// TwinCAT 3 PLC project RTNNI
// Title: Real-Time Neural Network generator
// Company: ISW
// Author: Zexu Zhou, Christoph Hinze
// ProjectVersion: 0.1
// ProgramVersion: 3.1.4024.0
// libraries:
//   Tc2_Standard, * (Beckhoff Automation GmbH)
//   Tc2_System, * (Beckhoff Automation GmbH)
//   Tc2_Utilities, * (Beckhoff Automation GmbH)
//   Tc3_Module, * (Beckhoff Automation GmbH)
// project tree:
//   DUTs/ act_type.TcDUT (not stored), Dense_v1_Layers.TcDUT, Dense_v1_LayerWeights.TcDUT, Layer.TcDUT (not stored), norm_type.TcDUT
//   / PlcTask.TcTTO
//   POUs/activation function/ F_exponential.TcPOU (not stored), F_relu.TcPOU (not stored), F_selu.TcPOU, F_sigmoid.TcPOU (not stored), F_silu.TcPOU (not stored), F_softplus.TcPOU, F_softsign.TcPOU (not stored), F_tanh.TcPOU
//   POUs/ FB_Dense_v1.TcPOU, FB_LoadWeights.TcPOU, F_ForwardPropagation.TcPOU (not stored), MAIN.TcPOU
//   POUs/math/ F_Dot.TcPOU (not stored)
//   POUs/normalization/ F_denormalization.TcPOU (not stored), F_normalization.TcPOU (not stored), F_NormalizationLayer.TcPOU

CONFIGURATION RTNNI
    RESOURCE PLC ON TwinCAT3
        TASK PlcTask(INTERVAL := T#10ms, PRIORITY := 21);
        PROGRAM MAIN WITH PlcTask : MAIN;
    END_RESOURCE
END_CONFIGURATION

// ---- DUTs/Dense_v1_Layers.TcDUT
TYPE Dense_v1_Layers:
STRUCT
    num_layers : UINT := 5;
    weights : Dense_v1_LayerWeights;
    layers : ARRAY[0..4] OF Layer :=[
    (num_neurons := 5),
    (num_neurons := 100, activation := act_type.relu, pointer_weight:= ADR(weights.HiddenLayers1_weight),pointer_bias:= ADR(weights.HiddenLayers1_bias)),
    (num_neurons := 100, activation := act_type.relu, pointer_weight:= ADR(weights.HiddenLayers2_weight),pointer_bias:= ADR(weights.HiddenLayers2_bias)),
    (num_neurons := 100, activation := act_type.relu, pointer_weight:= ADR(weights.HiddenLayers3_weight),pointer_bias:= ADR(weights.HiddenLayers3_bias)),
    (num_neurons := 1,activation := act_type.linear, normalization := norm_type.denormalization, pointer_weight:= ADR(weights.OutputLayer_weight),pointer_bias:= ADR(weights.OutputLayer_bias))];
    layer_output : ARRAY[0..99] OF LREAL;
    layer_input : ARRAY[0..99] OF LREAL;
    
END_STRUCT
END_TYPE

// ---- DUTs/Dense_v1_LayerWeights.TcDUT
TYPE Dense_v1_LayerWeights:
STRUCT
    normalization_mean : ARRAY[0..0] OF LREAL;
    normalization_std : ARRAY[0..0] OF LREAL;
    HiddenLayers1_weight : ARRAY[0..99,0..4] OF LREAL;
    HiddenLayers1_bias : ARRAY[0..99] OF LREAL;
    HiddenLayers2_weight : ARRAY[0..99,0..99] OF LREAL;
    HiddenLayers2_bias : ARRAY[0..99] OF LREAL;
    HiddenLayers3_weight : ARRAY[0..99,0..99] OF LREAL;
    HiddenLayers3_bias : ARRAY[0..99] OF LREAL;
    OutputLayer_weight : ARRAY[0..0,0..99] OF LREAL;
    OutputLayer_bias : ARRAY[0..0] OF LREAL;
    denormalization_mean : ARRAY[0..0] OF LREAL;
    denormalization_std : ARRAY[0..0] OF LREAL;
    hash_sha_256 : ARRAY[0..3] OF LREAL;
END_STRUCT
END_TYPE

// ---- DUTs/norm_type.TcDUT
{attribute 'qualified_only'}
{attribute 'strict'}
TYPE norm_type :
(	
	none := 0,	
	normalization := 1,
	denormalization :=2
);
END_TYPE

// ---- POUs/MAIN.TcPOU
PROGRAM MAIN
VAR
	input : ARRAY[0..4] OF LREAL := [1,1,1,1,1];	
	out : ARRAY[0..0] OF LREAL;
	FB_NN : FB_Dense_v1;
	
	test_in : LREAL := 50;
	test_flg : BOOL := FALSE;
END_VAR

FB_NN(pointer_input := ADR(input),pointer_output:= ADR(out));
IF NOT test_flg THEN
	F_NormalizationLayer(pointer_input := ADR(test_in),pointer_mean := ADR(FB_NN.nn.weights.denormalization_mean),
	pointer_std := ADR(FB_NN.nn.weights.denormalization_std),invert := TRUE, num_neurons := FB_NN.nn.layers[SIZEOF(FB_NN.nn.layers)/SIZEOF(FB_NN.nn.layers[0])-1].num_neurons);
	test_flg := TRUE;
END_IF

END_PROGRAM

// ---- POUs/FB_Dense_v1.TcPOU
FUNCTION_BLOCK FB_Dense_v1
VAR_INPUT
	pointer_input: POINTER TO LREAL;
	pointer_output : POINTER TO LREAL;
	
END_VAR
VAR	
  i : UINT;
  id : UINT;
  iq : UINT;
  flag_AreWeightsLoaded : BOOL := FALSE;
  flag_AreWeightsChecked : BOOL := FALSE;
  load_weights : FB_LoadWeights;
  filePath : T_MaxString := 'c:\Users\Administrator\Documents\git-projekte\keras2plc\tests\test_ST_files\Dense_v1_weights.dat';
  nn : Dense_v1_Layers;
  hash_sha_256_twincat : ARRAY[0..3] OF LREAL;
  compare_res : DINT := 99;
END_VAR

IF NOT flag_AreWeightsLoaded THEN
		load_weights(execute := TRUE,filePath := filePath,ReadAdr := ADR(nn.weights), ReadLen :=  SIZEOF(nn.weights));
		IF NOT load_weights.busy THEN 
			flag_AreWeightsLoaded := TRUE;
		END_IF
ELSIF NOT flag_AreWeightsChecked THEN
	F_GenerateHashValue(hashMode:=E_HashMode.HASH_SHA256,pData := ADR(nn.weights),nData := SIZEOF(nn.weights)-32,pHash := ADR(hash_sha_256_twincat),nHash:=32);
	compare_res := MEMCMp(pBuf1 := ADR(hash_sha_256_twincat),ADR(nn.weights.hash_sha_256),32);
	IF compare_res = 0 THEN
		flag_AreWeightsChecked := TRUE;
	END_IF
ELSE
	MEMCPY(destAddr:=ADR(nn.layer_input),srcAddr:=pointer_input,n:=SIZEOF(LREAL)*nn.layers[0].num_neurons);
  // input normalization
	IF nn.layers[0].normalization = norm_type.normalization THEN
		F_NormalizationLayer(pointer_input := ADR(nn.layer_input),pointer_mean := ADR(nn.weights.normalization_mean),
			pointer_std := ADR(nn.weights.normalization_std),invert := FALSE, num_neurons := nn.layers[0].num_neurons); 
	END_IF
  // forward inference
	FOR i := 0 TO nn.num_layers-2 DO
		F_ForwardPropagation(	layer_pre	:= 	nn.layers[i],
								layer_next	:=	nn.layers[i+1],
								pointer_in 	:=	ADR(nn.layer_input),
								pointer_out	:=	ADR(nn.layer_output)	);
		MEMCPY(destAddr:=ADR(nn.layer_input),srcAddr:=ADR(nn.layer_output),n:=SIZEOF(LREAL)*nn.layers[i+1].num_neurons);
	END_FOR
	MEMCPY(destAddr:=pointer_output,srcAddr:=ADR(nn.layer_output),n:=SIZEOF(LREAL)*nn.layers[SIZEOF(nn.layers)/SIZEOF(nn.layers[0])-1].num_neurons);
  // output denormalization
	IF nn.layers[SIZEOF(nn.layers)/SIZEOF(nn.layers[0])-1].normalization = norm_type.denormalization THEN
		F_NormalizationLayer(pointer_input := ADR(pointer_output),pointer_mean := ADR(nn.weights.denormalization_mean),
			pointer_std := ADR(nn.weights.denormalization_std),invert := TRUE, num_neurons := nn.layers[SIZEOF(nn.layers)/SIZEOF(nn.layers[0])-1].num_neurons);
	END_IF
END_IF

END_FUNCTION_BLOCK

// ---- POUs/FB_LoadWeights.TcPOU
FUNCTION_BLOCK FB_LoadWeights
VAR_INPUT
	execute : BOOL := FALSE;
	filePath : T_MaxString;
	ReadAdr :POINTER TO LREAL;
	ReadLen : UDINT;
END_VAR
VAR_OUTPUT
	busy : BOOL ;
END_VAR
VAR
	 
	i : UINT;
	step : UINT := 1;
	fbFileOpen : FB_FileOpen;
	hFile : UINT;
	fbFileRead : FB_FileRead;
	fbFileClose : FB_FileClose;
END_VAR

CASE step OF
	1:
		busy := FALSE;
		IF execute THEN
			step := step + 1;
			busy := TRUE;
		END_IF
	2: 
		fbFileOpen(bExecute := FALSE);
		fbFileOpen(sPathName := filePath ,nMode := FOPEN_MODEREAD OR FOPEN_MODEBINARY, bExecute := TRUE);
		step := step+1;
	3:
		fbFileOpen(bExecute := FALSE);
		IF NOT fbFileOpen.bBusy THEN
			hFile := fbFileOpen.hFile;
			step := step +1;
		END_IF
	4:
		fbFileRead(bExecute := FALSE);
		fbFileRead(hFile := hFile,pReadBuff := ReadAdr ,cbReadLen := ReadLen,bEXecute := TRUE);
		step := step +1;
	5:
		fbFileRead(bExecute := FALSE);
		IF NOT fbFileRead.bBusy THEN
			fbFileClose(bExecute := FALSE);		
			fbFileClose(hFile:= hFile, bExecute := TRUE);
			step := step +1;
		END_IF
	6:
		fbFileClose(bExecute := FALSE);	
		IF NOT fbFileClose.bBusy THEN
			step := 1;
			busy := FALSE;
			execute := FALSE;
		END_IF
END_CASE

END_FUNCTION_BLOCK

// ---- POUs/normalization/F_NormalizationLayer.TcPOU
FUNCTION F_NormalizationLayer : BOOL
VAR_INPUT
	pointer_input : POINTER TO LREAL;
	pointer_mean : POINTER TO LREAL;
	pointer_std : POINTER TO LREAL;
	invert: BOOL;
	num_neurons : UINT;
END_VAR
VAR
	in : UINT;
	id : UINT;
END_VAR

IF NOT invert THEN
	FOR in := 0 TO num_neurons-1 DO
		pointer_input[in] := F_normalization(x:=pointer_input[in],mean:=pointer_mean[in],std:=pointer_std[in]);
	END_FOR
ELSE
	FOR id := 0 TO num_neurons-1 DO
		 pointer_input[id] := F_denormalization(x:=pointer_input[id],mean:=pointer_mean[id],std:=pointer_std[id]);
	END_FOR
END_IF

END_FUNCTION

// ---- POUs/activation function/F_selu.TcPOU
FUNCTION F_selu : lreal
VAR_INPUT
	x : LREAL;
END_VAR
VAR
	scale : LREAL := 1.05070098;
	alpha : LREAL := 1.67326324;
END_VAR

IF x > 0 THEN
	F_selu := scale * x;
ELSIF x < -1E2 THEN
	F_selu := - scale * alpha;
ELSE
	F_selu := scale * alpha * (exp(x) - 1);
END_IF

END_FUNCTION

// ---- POUs/activation function/F_softplus.TcPOU
FUNCTION F_softplus : lreal
VAR_INPUT
	x : LREAL;
END_VAR

IF x > 1E2 THEN
	F_softplus := x;
ELSIF x < -1E2 THEN
	F_softplus := 0;
ELSE
	F_softplus := LOG(EXP(x)+1);
END_IF

END_FUNCTION

// ---- POUs/activation function/F_tanh.TcPOU
FUNCTION F_tanh : LREAL
VAR_INPUT
	x: LREAL;
END_VAR

IF x > 1E2 THEN
	F_tanh := 1;
ELSIF x < -1E2 THEN
	F_tanh := -1;
ELSE
	F_tanh := (EXP(x) - EXP(-x))/(EXP(x) + EXP(-x));
END_IF

END_FUNCTION
